{attribute addProperty BoxType "EK1122-0000-0018"}
{attribute addProperty Id "Beckhoff_EKM1xxxsub_EK1100EK1100_179A0949162A_0001_EKM1101_0000_0016EKM1101_CC1E967461977.375A_0002_EKM1101_0000_0017EKM1101_CC1E967461977.375A_0003_EKM1101_0000_0018EKM1101_CC1E967461977.375A_0004_EKM1101_0000_0019EKM1101_87969BFD51464.25A_0005_EKM1101_0000_0020EKM1101_87969BFD51464.25"}
{attribute addProperty CRC "3624566892"}
{attribute addProperty SizeInBites "2901"}
{attribute addProperty SizeInBytes "362.625"}
TYPE Beckhoff_EKM1xxxEK1122_D80A806C EXTENDS EK1122_179A0949 :
STRUCT
	{attribute addProperty Name "Beckhoff_EKM1xxxsub_EK1100"}
	Beckhoff_EKM1xxxsub_EK1100 : EK1100_179A0949;
	{attribute addProperty Name "A_0001_EKM1101_0000_0016"}
	A_0001_EKM1101_0000_0016 : EKM1101_CC1E9674;
	{attribute addProperty Name "A_0002_EKM1101_0000_0017"}
	A_0002_EKM1101_0000_0017 : EKM1101_CC1E9674;
	{attribute addProperty Name "A_0003_EKM1101_0000_0018"}
	A_0003_EKM1101_0000_0018 : EKM1101_CC1E9674;
	{attribute addProperty Name "A_0004_EKM1101_0000_0019"}
	A_0004_EKM1101_0000_0019 : EKM1101_87969BFD;
	{attribute addProperty Name "A_0005_EKM1101_0000_0020"}
	A_0005_EKM1101_0000_0020 : EKM1101_87969BFD;
END_STRUCT
END_TYPE

(* stored: Version 1.2.0.0, ProductVersion 3.1.4024.9
   DUT Beckhoff_EKM1xxxEK1122_D80A806C: Id {007c2d5f-0968-42cb-9811-87cdfa24a43a} *)
